(* PLC project Unnamed, Unknown Unnamed 1 *)
(* stored: creationDateTime 2013-01-29T14:01:00, modificationDateTime 2013-04-04T11:06:06 *)

PROGRAM program0
  VAR
    beat : BOOL;
    count : INT;
    LOGGER0 : LOGGER;
    lvl : LOGLEVEL := WARNING;
  END_VAR
  VAR  (* added by the conversion: wires and edge detectors of the diagram *)
    _NOT3_OUT : BOOL;
    R_TRIG1 : R_TRIG;
    _ADD5_OUT : INT;
  END_VAR

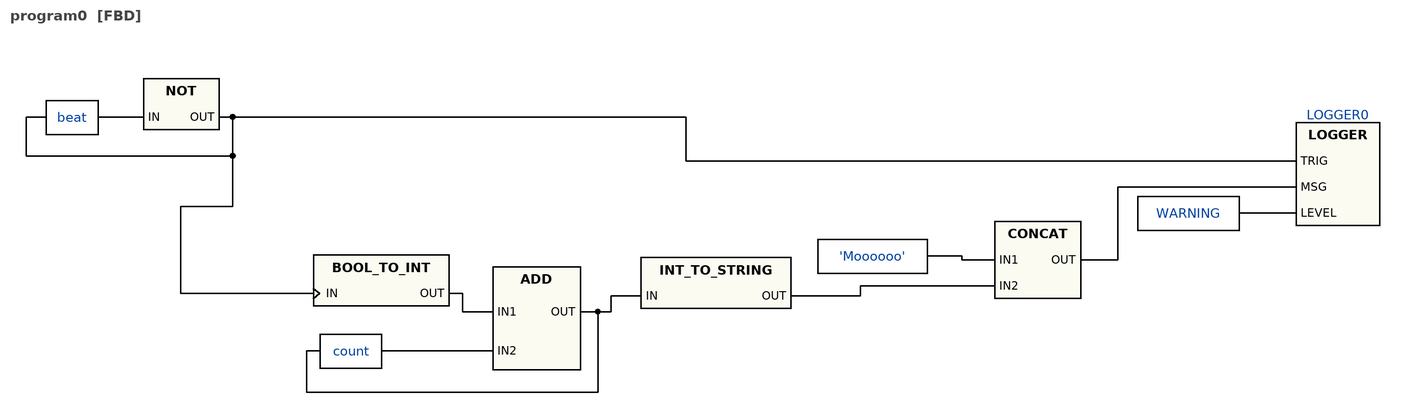
(* FBD diagram, written out as Structured Text *)
_NOT3_OUT := NOT beat;
beat := _NOT3_OUT;
R_TRIG1(CLK := _NOT3_OUT);
_ADD5_OUT := BOOL_TO_INT(R_TRIG1.Q) + count;
count := _ADD5_OUT;
LOGGER0(TRIG := _NOT3_OUT, MSG := CONCAT('Moooooo', INT_TO_STRING(_ADD5_OUT)), LEVEL := WARNING);
END_PROGRAM

CONFIGURATION config
  RESOURCE resource1 ON PLC
    TASK blob(INTERVAL := T#100ms, PRIORITY := 0);
    PROGRAM blub WITH blob : program0;
  END_RESOURCE
END_CONFIGURATION
